// TIA Portal V18 export
DATA_BLOCK "Temperature_DB"   // DB7
VERSION : 0.1
// stored: AutoNumber true, InstanceOfName Temperature, InstanceOfType FB
"Temperature"
BEGIN
END_DATA_BLOCK
